(* IEC 61131-3 sources: ax-factoryio-assembler/src/component, 6 files *)

(* ---- OperationMode.st ---- *)
TYPE
    OperationMode : (Manual, Auto);
END_TYPE

CLASS ModeSwitch
    VAR PRIVATE
        _mode: OperationMode;
    END_VAR

    METHOD PUBLIC GetOperationMode: OperationMode
        GetOperationMode := _mode;
    END_METHOD

    METHOD PUBLIC Input
        VAR_INPUT
            Auto:BOOL;
        END_VAR

        IF Auto THEN
            _mode := OperationMode#Auto;
        ELSE
            _mode := OperationMode#Manual;
        END_IF;
    END_METHOD
END_CLASS

(* ---- TwoAxisPickPlace.st ---- *)
USING System.Timer;

TYPE
    PickPlaceStatus : (
IDLE,
        READY,
        PICK_MOVING_Z_DOWN,
        GRABING,
        PICK_MOVING_Z_UP,
        MOVING_X_RIGHT,
        PLACE_MOVING_Z_DOWN,
        RELEASE,
        PLACE_MOVING_Z_UP,
        DONE);
END_TYPE

CLASS TwoAxisPickPlace
    VAR
        _moveZCmd : BOOL;
        _movingZ : BOOL;
        _moveXCmd : BOOL;
        _movingX : BOOL;
        _grabCmd : BOOL;
        _itemDetected : BOOL;
        _status : PickPlaceStatus;
        _delayTimer : OnDelay;
    END_VAR

    METHOD PUBLIC Input
        VAR_INPUT
            movingX : BOOL;
            movingZ : BOOL;
            itemDetected : BOOL;
        END_VAR
        _movingX := movingX;
        _movingZ := movingZ;
        _itemDetected := itemDetected;
    END_METHOD

    METHOD PUBLIC Output
        VAR_OUTPUT
            qMoveX : BOOL;
            qMoveZ : BOOL;
            qGrab : BOOL;
        END_VAR
        qMoveX := _moveXCmd;
        qMoveZ := _moveZCmd;
        qGrab := _grabCmd;
    END_METHOD

    METHOD PUBLIC Start
        _status := PickPlaceStatus#READY;
    END_METHOD

    METHOD PUBLIC Cycle
        CASE _status OF
            PickPlaceStatus#IDLE:
                ;
            PickPlaceStatus#READY:
                _moveZCmd := TRUE;
                _status := PickPlaceStatus#PICK_MOVING_Z_DOWN;
                _delayTimer(FALSE);
            PickPlaceStatus#PICK_MOVING_Z_DOWN:
                _delayTimer(NOT (_movingZ), LT#200ms);
                IF _delayTimer.output THEN
                    _delayTimer(FALSE);
                    _grabCmd := TRUE;
                    _status := PickPlaceStatus#GRABING;
                END_IF;
            PickPlaceStatus#GRABING:
                _delayTimer(_itemDetected, LT#200ms);
                IF _delayTimer.output THEN
                    _moveZCmd := FALSE;
                    _delayTimer(FALSE);
                    _status := PickPlaceStatus#PICK_MOVING_Z_UP;
                END_IF;
            PickPlaceStatus#PICK_MOVING_Z_UP:
                _delayTimer(NOT (_movingZ), LT#200ms);
                IF _delayTimer.output THEN
                    _moveXCmd := TRUE;
                    _delayTimer(FALSE);
                    _status := PickPlaceStatus#MOVING_X_RIGHT;
                END_IF;
            PickPlaceStatus#MOVING_X_RIGHT:
                _delayTimer(NOT (_movingX), LT#200ms);
                IF _delayTimer.output THEN
                    _moveZCmd := TRUE;
                    _delayTimer(FALSE);
                    _status := PickPlaceStatus#PLACE_MOVING_Z_DOWN;
                END_IF;
            PickPlaceStatus#PLACE_MOVING_Z_DOWN:
                _delayTimer(NOT (_movingZ), LT#200ms);
                IF _delayTimer.output THEN
                    _moveZCmd := FALSE;
                    _grabCmd := FALSE;
                    _delayTimer(FALSE);
                    _status := PickPlaceStatus#PLACE_MOVING_Z_UP;
                END_IF;
            PickPlaceStatus#PLACE_MOVING_Z_UP:
                _moveXCmd := FALSE;
                _status := PickPlaceStatus#DONE;
            PickPlaceStatus#DONE:
                _moveZCmd := FALSE;
                _moveXCmd := FALSE;
                _grabCmd := FALSE;
        END_CASE;
    END_METHOD

    METHOD PUBLIC Reset
        _moveZCmd := FALSE;
        _moveXCmd := FALSE;
        _grabCmd := FALSE;
        _status := PickPlaceStatus#READY;
    END_METHOD

    METHOD PUBLIC IsDone : BOOL
        IsDone := (_status = PickPlaceStatus#DONE);
    END_METHOD
END_CLASS

(* ---- Button.st ---- *)
CLASS Button
    VAR PRIVATE
        _isPressed : BOOL;
    END_VAR

    METHOD PUBLIC IsPressed : BOOL
        ;
        IsPressed := _isPressed;
    END_METHOD

    METHOD PUBLIC Cycle
        VAR_INPUT
            ButtonInputSignal : BOOL;
        END_VAR
        _isPressed := ButtonInputSignal;
    END_METHOD
END_CLASS

CLASS ButtonWithLight
    VAR PRIVATE
        _isPressed : BOOL;
    END_VAR

    METHOD PUBLIC IsPressed : BOOL
        ;
        IsPressed := _isPressed;
    END_METHOD

    METHOD PUBLIC Input
        VAR_INPUT
            ButtonInputSignal : BOOL;
        END_VAR
        _isPressed := ButtonInputSignal;
    END_METHOD

    METHOD PUBLIC Output
        VAR_OUTPUT
            ButtonLightOutputSignal : BOOL;
        END_VAR
        ButtonLightOutputSignal := _isPressed;
    END_METHOD
END_CLASS

(* ---- Clamp.st ---- *)
CLASS Clamp
    VAR
        _clampCmd : BOOL;
        _clamped : BOOL;
    END_VAR

    METHOD PUBLIC Input
        VAR_INPUT
            clamped : BOOL;
        END_VAR
        _clamped := clamped;
    END_METHOD

    METHOD PUBLIC Output
        VAR_OUTPUT
            clamp : BOOL;
        END_VAR
        clamp := _clampCmd;
    END_METHOD

    METHOD IsClamped : BOOL
        IsClamped := _clamped;
    END_METHOD

    METHOD PUBLIC DoClamp
        _clampCmd := TRUE;
    END_METHOD

    METHOD PUBLIC Release
        _clampCmd := FALSE;
    END_METHOD
END_CLASS

(* ---- Conveyor.st ---- *)
USING System.Timer;

CLASS Conveyor
    VAR
        _isOn : BOOL;
        _isStopped : BOOL;
        _stopTimer: OnDelay;
        _elapsedTime: LTIME;
    END_VAR

    METHOD PUBLIC Start
        _isOn := TRUE;
    END_METHOD

    METHOD PUBLIC Stop
        _isOn := FALSE;
    END_METHOD

    METHOD IsStopped : BOOL
        IsStopped := NOT(_isOn);
    END_METHOD

    METHOD PUBLIC Output
        VAR_OUTPUT
            run : BOOL;
        END_VAR
        run := _isOn;
    END_METHOD
END_CLASS

(* ---- Sensor.st ---- *)
CLASS ObjectSensor
    VAR
        _hasObjectPassed: BOOL;
    END_VAR

    METHOD PUBLIC Input : Int
        VAR_INPUT
            objectDetectedInput: BOOL;
        END_VAR

        _hasObjectPassed :=  _hasObjectPassed | objectDetectedInput;
    END_METHOD

    METHOD PUBLIC HasObjectPassed : BOOL
        HasObjectPassed := _hasObjectPassed;
    END_METHOD

    METHOD PUBLIC Reset
        _hasObjectPassed :=FALSE;
    END_METHOD
END_CLASS
